PROGRAM MotionCtrl
VAR
END_VAR

SingleAxis_LD();

METHOD SingleAxis_LD : BOOL
VAR_INPUT
END_VAR
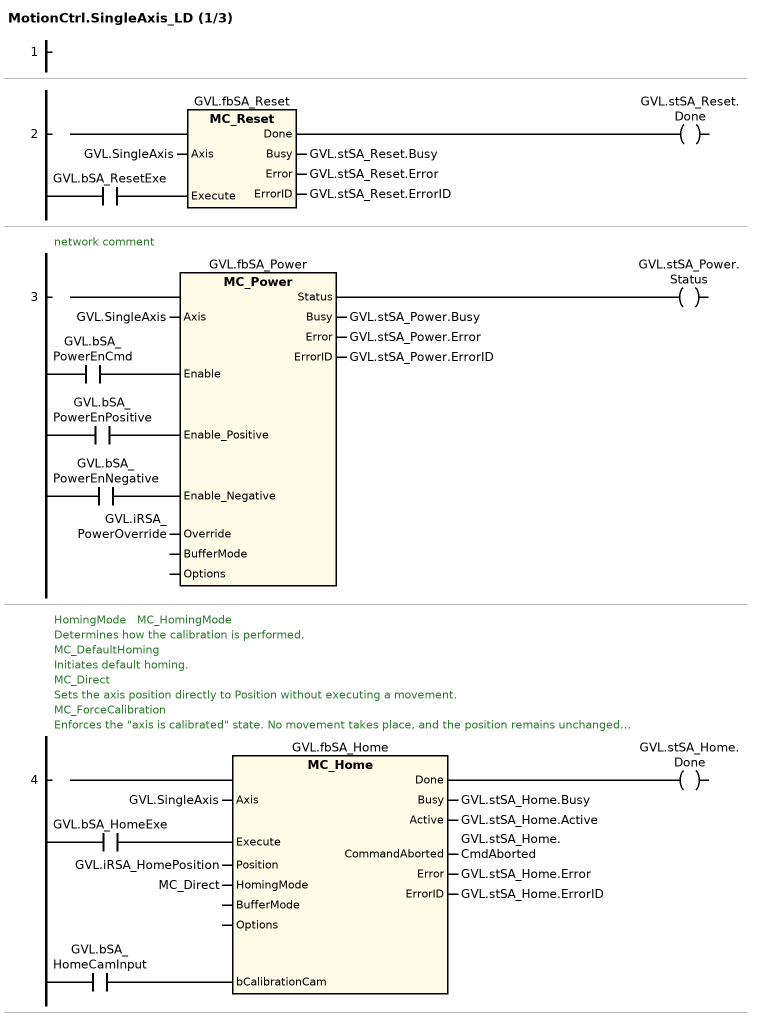
// NETWORK 1

// NETWORK 2
GVL.fbSA_Reset(
    Axis := GVL.SingleAxis,
    Execute := GVL.bSA_ResetExe,
    Busy => GVL.stSA_Reset.Busy,
    Error => GVL.stSA_Reset.Error,
    ErrorID => GVL.stSA_Reset.ErrorID); // MC_Reset
GVL.stSA_Reset.Done := GVL.fbSA_Reset.Done;

// NETWORK 3
// network comment
GVL.fbSA_Power(
    Axis := GVL.SingleAxis,
    Enable := GVL.bSA_PowerEnCmd,
    Enable_Positive := GVL.bSA_PowerEnPositive,
    Enable_Negative := GVL.bSA_PowerEnNegative,
    Override := GVL.iRSA_PowerOverride,
    Busy => GVL.stSA_Power.Busy,
    Error => GVL.stSA_Power.Error,
    ErrorID => GVL.stSA_Power.ErrorID); // MC_Power
GVL.stSA_Power.Status := GVL.fbSA_Power.Status;

// NETWORK 4
// HomingMode   MC_HomingMode
// Determines how the calibration is performed.
//
// MC_DefaultHoming
// Initiates default homing.
// MC_Direct
// Sets the axis position directly to Position without executing a movement.
// MC_ForceCalibration
// Enforces the "axis is calibrated" state. No movement takes place, and the position remains unchanged.
// MC_ResetCalibration
// Resets the calibration state of the axis. No movement takes place, and the position remains unchanged.
GVL.fbSA_Home(
    Axis := GVL.SingleAxis,
    Execute := GVL.bSA_HomeExe,
    Position := GVL.iRSA_HomePosition,
    HomingMode := MC_Direct,
    bCalibrationCam := GVL.bSA_HomeCamInput,
    Busy => GVL.stSA_Home.Busy,
    Active => GVL.stSA_Home.Active,
    CommandAborted => GVL.stSA_Home.CmdAborted,
    Error => GVL.stSA_Home.Error,
    ErrorID => GVL.stSA_Home.ErrorID); // MC_Home
GVL.stSA_Home.Done := GVL.fbSA_Home.Done;

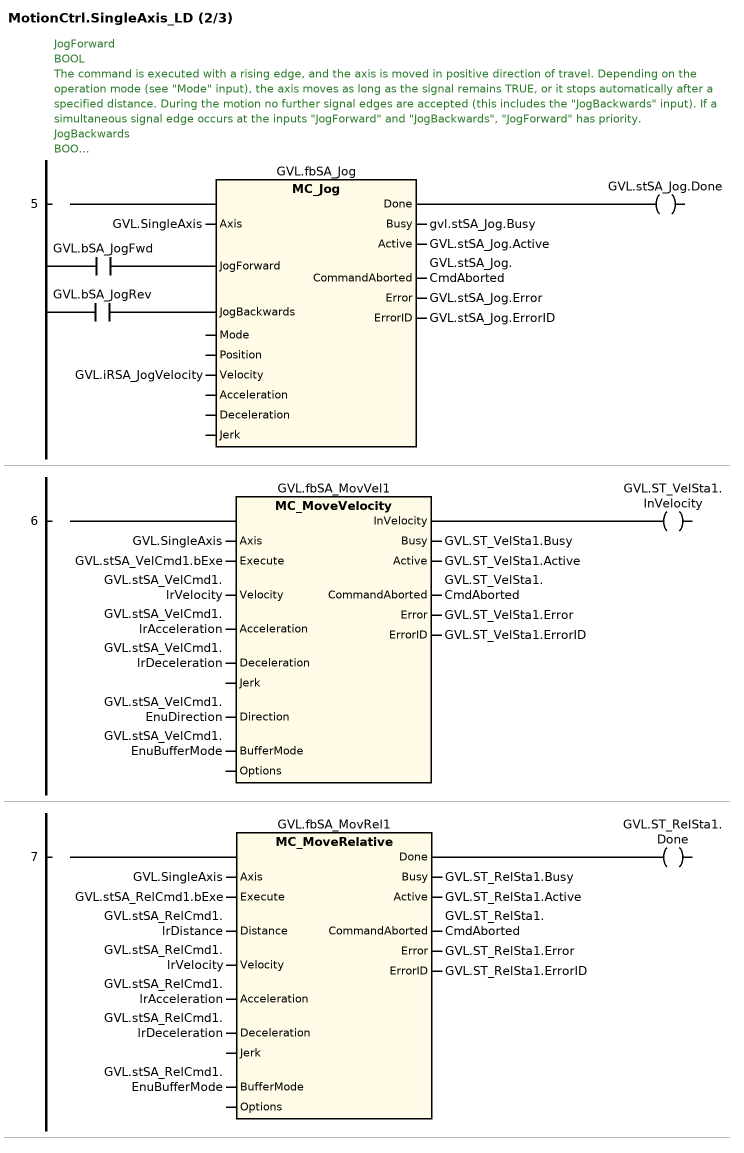
// NETWORK 5
// JogForward
//
// BOOL
//
// The command is executed with a rising edge, and the axis is moved in positive direction of travel. Depending on the operation mode (see "Mode" input), the axis moves as long as the signal remains TRUE, or it stops automatically after a specified distance. During the motion no further signal edges are accepted (this includes the "JogBackwards" input). If a simultaneous signal edge occurs at the inputs "JogForward" and "JogBackwards", "JogForward" has priority.
//
// JogBackwards
//
// BOOL
//
// The command is executed with a rising edge, and the axis is moved in negative direction of travel. "JogForward" and "JogBackwards" should be triggered alternatively, although they are also mutually locked internally.
//
// Mode
//
// E_JogMode
//
// Determines the operation mode in which the manual function is executed.
//
// MC_JOGMODE_STANDARD_SLOW
// the axis moves as long as the signal at one of the jog inputs is TRUE. The "low velocity for manual functions" specified in the TwinCAT System Manager and standard dynamics are used. In this operation mode the position, velocity and dynamics data specified in the function block have no effect.
// MC_JOGMODE_STANDARD_FAST
// the axis moves as long as the signal at one of the jog inputs is TRUE. The "high velocity for manual functions" specified in the TwinCAT System Manager and standard dynamics are used. In this operation mode the position, velocity and dynamics data specified in the function block have no effect.
// MC_JOGMODE_CONTINUOUS
// The axis moves as long as the signal at one of the jog inputs is TRUE. The velocity and dynamics data specified by the user are used. The position has no effect.
// MC_JOGMODE_INCHING
// With a rising edge at one of the jog inputs the axis is moved by a certain distance which is specified via the "Position" input. The axis stops automatically, irrespective of the state of the jog inputs. A new movement step is only executed once a further rising edge is encountered. With each start the velocity and dynamics data specified by the user are used.
// MC_JOGMODE_INCHING_MODULO
// With a rising edge at one of the jog inputs the axis is moved by a certain distance which is specified via the "Positions" input. The axis position will snap to an integer multiple of the position parameter. The axis stops automatically, irrespective of the state of the jog inputs. A new movement step is only executed once a further rising edge is encountered. With each start the velocity and dynamics data specified by the user are used.
// Position
//
// LREAL
//
// Relative distance for movements in MC_JOGMODE_INCHING operation mode.
//
// Velocity
//
// LREAL
//
// Maximum travel velocity (>0).
//
// Acceleration
//
// LREAL
//
// Acceleration (≥0). If the value is 0, the standard acceleration from the axis configuration in the System Manager is used.
//
// Deceleration
//
// LREAL
//
// Deceleration (≥0). If the value is 0, the standard deceleration from the axis configuration in the System Manager is used.
//
// Jerk
//
// LREAL
//
// Jerk (≥0). At a value of 0, the standard jerk from the axis configuration in the System Manager is applied.
GVL.fbSA_Jog(
    Axis := GVL.SingleAxis,
    JogForward := GVL.bSA_JogFwd,
    JogBackwards := GVL.bSA_JogRev,
    Velocity := GVL.iRSA_JogVelocity,
    Busy => gvl.stSA_Jog.Busy,
    Active => GVL.stSA_Jog.Active,
    CommandAborted => GVL.stSA_Jog.CmdAborted,
    Error => GVL.stSA_Jog.Error,
    ErrorID => GVL.stSA_Jog.ErrorID); // MC_Jog
GVL.stSA_Jog.Done := GVL.fbSA_Jog.Done;

// NETWORK 6
GVL.fbSA_MovVel1(
    Axis := GVL.SingleAxis,
    Execute := GVL.stSA_VelCmd1.bExe,
    Velocity := GVL.stSA_VelCmd1.lrVelocity,
    Acceleration := GVL.stSA_VelCmd1.lrAcceleration,
    Deceleration := GVL.stSA_VelCmd1.lrDeceleration,
    Direction := GVL.stSA_VelCmd1.EnuDirection,
    BufferMode := GVL.stSA_VelCmd1.EnuBufferMode,
    Busy => GVL.ST_VelSta1.Busy,
    Active => GVL.ST_VelSta1.Active,
    CommandAborted => GVL.ST_VelSta1.CmdAborted,
    Error => GVL.ST_VelSta1.Error,
    ErrorID => GVL.ST_VelSta1.ErrorID); // MC_MoveVelocity
GVL.ST_VelSta1.InVelocity := GVL.fbSA_MovVel1.InVelocity;

// NETWORK 7
GVL.fbSA_MovRel1(
    Axis := GVL.SingleAxis,
    Execute := GVL.stSA_RelCmd1.bExe,
    Distance := GVL.stSA_RelCmd1.lrDistance,
    Velocity := GVL.stSA_RelCmd1.lrVelocity,
    Acceleration := GVL.stSA_RelCmd1.lrAcceleration,
    Deceleration := GVL.stSA_RelCmd1.lrDeceleration,
    BufferMode := GVL.stSA_RelCmd1.EnuBufferMode,
    Busy => GVL.ST_RelSta1.Busy,
    Active => GVL.ST_RelSta1.Active,
    CommandAborted => GVL.ST_RelSta1.CmdAborted,
    Error => GVL.ST_RelSta1.Error,
    ErrorID => GVL.ST_RelSta1.ErrorID); // MC_MoveRelative
GVL.ST_RelSta1.Done := GVL.fbSA_MovRel1.Done;

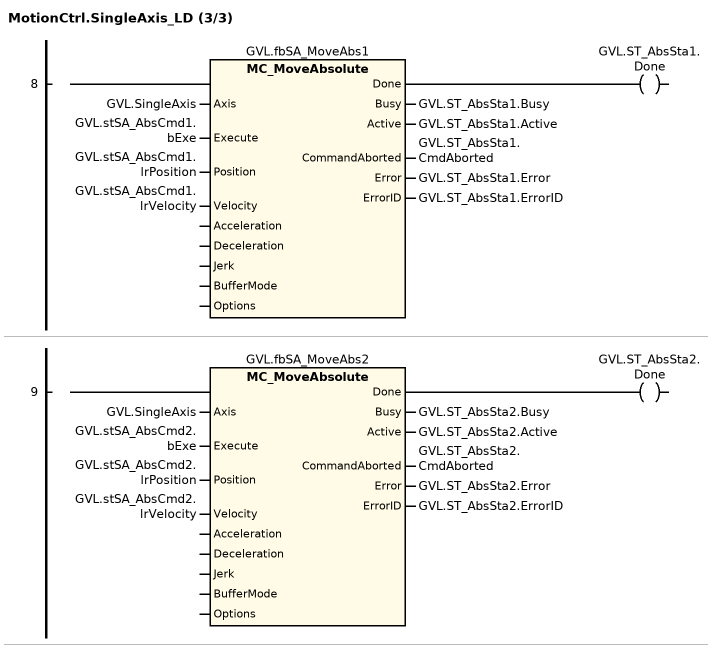
// NETWORK 8
GVL.fbSA_MoveAbs1(
    Axis := GVL.SingleAxis,
    Execute := GVL.stSA_AbsCmd1.bExe,
    Position := GVL.stSA_AbsCmd1.lrPosition,
    Velocity := GVL.stSA_AbsCmd1.lrVelocity,
    Busy => GVL.ST_AbsSta1.Busy,
    Active => GVL.ST_AbsSta1.Active,
    CommandAborted => GVL.ST_AbsSta1.CmdAborted,
    Error => GVL.ST_AbsSta1.Error,
    ErrorID => GVL.ST_AbsSta1.ErrorID); // MC_MoveAbsolute
GVL.ST_AbsSta1.Done := GVL.fbSA_MoveAbs1.Done;

// NETWORK 9
GVL.fbSA_MoveAbs2(
    Axis := GVL.SingleAxis,
    Execute := GVL.stSA_AbsCmd2.bExe,
    Position := GVL.stSA_AbsCmd2.lrPosition,
    Velocity := GVL.stSA_AbsCmd2.lrVelocity,
    Busy => GVL.ST_AbsSta2.Busy,
    Active => GVL.ST_AbsSta2.Active,
    CommandAborted => GVL.ST_AbsSta2.CmdAborted,
    Error => GVL.ST_AbsSta2.Error,
    ErrorID => GVL.ST_AbsSta2.ErrorID); // MC_MoveAbsolute
GVL.ST_AbsSta2.Done := GVL.fbSA_MoveAbs2.Done;
END_METHOD

END_PROGRAM

(* stored: Version 1.1.0.1, ProductVersion 3.1.4024.12
   POU MotionCtrl: Id {0ca4e378-32f6-480e-bab1-17b9586cf081}, SpecialFunc None
   Method SingleAxis_LD: Id {f1cfecdb-67dc-4204-acda-584e95b3849d} *)
